Yaskawa INFORM job: PA.JBI

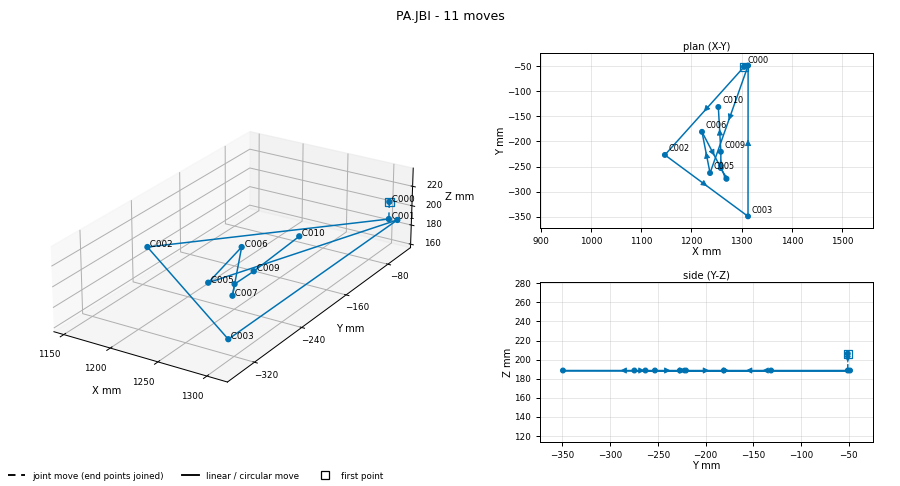
[picture p0: tool path of PA.JBI, 11 of 11 moves have a stored position in this frame; points joined in program order, loops and branches not executed]
/JOB
//NAME PA
//POS
///NPOS 11,0,0,0
///TOOL 0
///RECTAN
///RCONF 0,0,0,0,0
C000=1304.952,-51.025,206.350,-168.80,-11.35,-67.97
C001=1305.004,-51.000,188.655,-168.81,-11.35,-67.96
C002=1146.998,-226.882,188.630,-168.80,-11.35,-67.96
C003=1312.696,-349.303,188.655,-168.80,-11.35,-67.96
C004=1312.888,-48.655,188.655,-168.80,-11.35,-67.94
C005=1237.002,-262.934,188.655,-168.78,-11.34,-67.97
C006=1220.933,-180.827,188.655,-168.79,-11.36,-67.95
C007=1269.822,-274.516,188.655,-168.76,-11.35,-67.97
C008=1258.480,-252.974,188.655,-168.75,-11.34,-67.99
C009=1258.561,-220.551,188.655,-168.75,-11.34,-67.98
C010=1253.514,-131.331,188.655,-168.75,-11.33,-67.99
//INST
///DATE 2014/11/01 23:17
///ATTR 0,0,0,0,0,0,0,0,0,0,0,0,1,1,0,0
///FRAME BASE
NOP
*2
PAUSE
MOVJ C000 VJ=25.00 CONT
MOVJ C001 VJ=25.00 CONT
MOVL C002 V=375.0 CONT
MOVL C003 V=375.0 CONT
MOVL C004 V=375.0 CONT
MOVL C005 V=375.0 CONT
MOVL C006 V=375.0 CONT
MOVL C007 V=375.0 CONT
MOVL C008 V=375.0 CONT
MOVL C009 V=375.0 CONT
MOVL C010 V=375.0 CONT
JUMP *2
END
